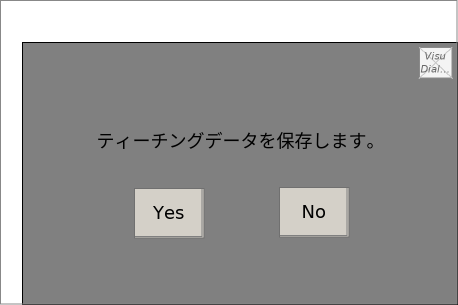
VISUALIZATION d_saveSample  // 458x305
    Rectangle (22,42 436x263)
    Image (419,47 33x31), image: VisuDialogs.ImagePoolDialogs.Delete
        OnMouseClick: CloseDialog Dialog=d_saveSample, Result=OK, NumpadKeypadSet=True
    Label (39,112 403x59), "ティーチングデータを保存します。"
    Button (134,188 70x50), "Yes"
        tap gvl_visu.flg_btn_saveSample
        OnMouseClick: CloseDialog Dialog=d_saveSample, Result=OK, NumpadKeypadSet=True
    Button (279,187 70x50), "No"
        OnMouseClick: CloseDialog Dialog=d_saveSample, Result=OK, NumpadKeypadSet=True
END_VISUALIZATION

(* stored: Version 1.1.0.1, ProductVersion 3.1.4024.12
   Visu d_saveSample: Id {049e68b7-087c-4f1d-b69d-0d431fe0dee4} *)
